(* CODESYS project date.and.time.190523.1.project

Project tree, tasks and I/O mapping:
  MIC7001 : Changsha Xiangji-ARM Cortex A9(xilinx zynq7000)-linux, Changsha Xiangji Hiden Technology Co.Ltd, version 3.5.10.40
    application Application
      libraries: Standard, * (System); CAA File, * (CAA Technical Workgroup); CAA Types Extern, * (CAA Technical Workgroup); CAA Callback Extern, * (CAA Technical Workgroup); SysMem, * (System); Util, 3.5.11.0 (System); SysFile, 3.5.9.0 (System); SysTypes Interfaces, * (System); CAN API, 1.0.0.3 (3S - Smart Software Solutions GmbH); AC_DataLog, 3.5.12.0 (3S - Smart Software Solutions GmbH); SysTime, * (System); CAA DTUtil Extern, 3.5.12.0 (CAA Technical Workgroup); CAA SerialCom, 3.5.12.0 (CAA Technical Workgroup); cyber gpio, 3.5.10.40 (cyber)
      task MainTask (cyclic, interval 20 ms, priority 15) calls prg_dateandtime
      DateAndTime/
        program prg_dateandtime [ST]
    SoftMotion General Axis Pool
  text list GlobalTextList
*)

// MIC7001/Application/DateAndTime/prg_dateandtime
PROGRAM prg_dateandtime
VAR
	new_DT : DATE_AND_TIME;
	dtu_get_dt : dtu.GetDateAndTime;	
	dtu_set_dt : dtu.SetDateAndTime;	
	
	//如果需要更改系统时间，请修改下列变量
	bTime_min: BYTE := 26;
	bTime_sec: BYTE := 23;
	bTime_hour: BYTE := 19;
	bTime_date: BYTE := 23;
	bTime_month: BYTE := 5;
	bTime_year: BYTE := 19;  //2019 只需要写19，程序会自动加上2000
	
	str_dt: STRING(255);

	f_set_dt:BOOL := FALSE;
END_VAR


//将f_set_dt 设置为 true，则自动修改系统时间，修改成功后 f_set_dt会自动变为false
IF f_set_dt THEN
	str_dt := concat('dt#', ANY_TO_STRING(2000+bTime_year));
	str_dt := concat(str_dt, '-');
	str_dt := concat(str_dt, ANY_TO_STRING(bTime_month));
	str_dt := concat(str_dt, '-');
	str_dt := concat(str_dt, ANY_TO_STRING(bTime_date));
	str_dt := concat(str_dt, '-');
	str_dt := concat(str_dt, ANY_TO_STRING(bTime_hour));
	str_dt := concat(str_dt, ':');
	str_dt := concat(str_dt, ANY_TO_STRING(bTime_min));
	str_dt := concat(str_dt, ':');
	str_dt := concat(str_dt, ANY_TO_STRING(bTime_sec));
	dtu_set_dt.dtDateAndTime := STRING_TO_DT(str_dt);

	dtu_set_dt(xExecute := FALSE);
	f_set_dt := FALSE;
END_IF
dtu_set_dt(xExecute := TRUE);

//读取系统时间，每个周期一次， new_DT中存放最新的时间
dtu_get_dt(xexecute := FALSE);
dtu_get_dt(xexecute := TRUE);

IF dtu_get_dt.xDone THEN
	new_DT := dtu_get_dt.dtDateAndTime;
END_IF

END_PROGRAM
